// SIMATIC S7-200 project (STEP 7-Micro/WIN), CPU 224XP REL 02.01

ORGANIZATION_BLOCK PRINCIPAL:OB1
TITLE=COMENTARIOS DEL PROGRAMA
BEGIN
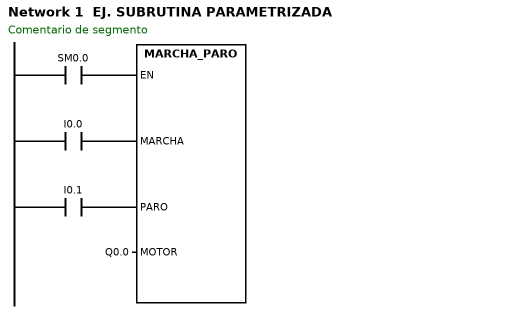
Network 1 // EJ. SUBRUTINA PARAMETRIZADA
// Comentario de segmento
// (network saved uncompiled; LAD cells follow)
// row 0: c0 -| |- SM0.0  c1 [MARCHA_PARO EN:=power@row0, MARCHA:=power@row1, PARO:=power@row2, MOTOR:=Q0.0]
// row 1: c0 -| |- I0.0  c1 [box]
// row 2: c0 -| |- I0.1  c1 [box]
// row 3: c1 [box]
END_ORGANIZATION_BLOCK

SUBROUTINE_BLOCK MARCHA_PARO:SBR0
TITLE=COMENTARIOS DE LA SUBRUTINA
VAR_INPUT
MARCHA:BOOL;	// L0.0 PURSTA EN MARCHA
PARO:BOOL;	// L0.1 REPOSO
END_VAR
VAR_IN_OUT
MOTOR:BOOL;	// L0.2 ARANQUE
END_VAR
BEGIN
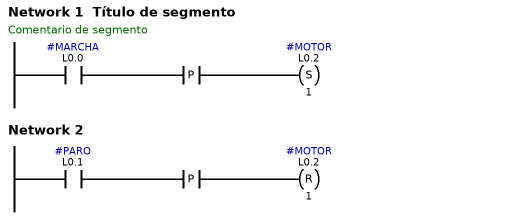
Network 1 // Título de segmento
// Comentario de segmento
// (network saved uncompiled; LAD cells follow)
// row 0: c0 -| |- #MARCHA:L0.0  c1 -|P|-  c2 -(S) #MOTOR:L0.2, 1
Network 2
// (network saved uncompiled; LAD cells follow)
// row 0: c0 -| |- #PARO:L0.1  c1 -|P|-  c2 -(R) #MOTOR:L0.2, 1
END_SUBROUTINE_BLOCK
